// Mitsubishi GX Works2 project: main_01   PLC: FX3U/FX3UC

PROGRAM MAIN
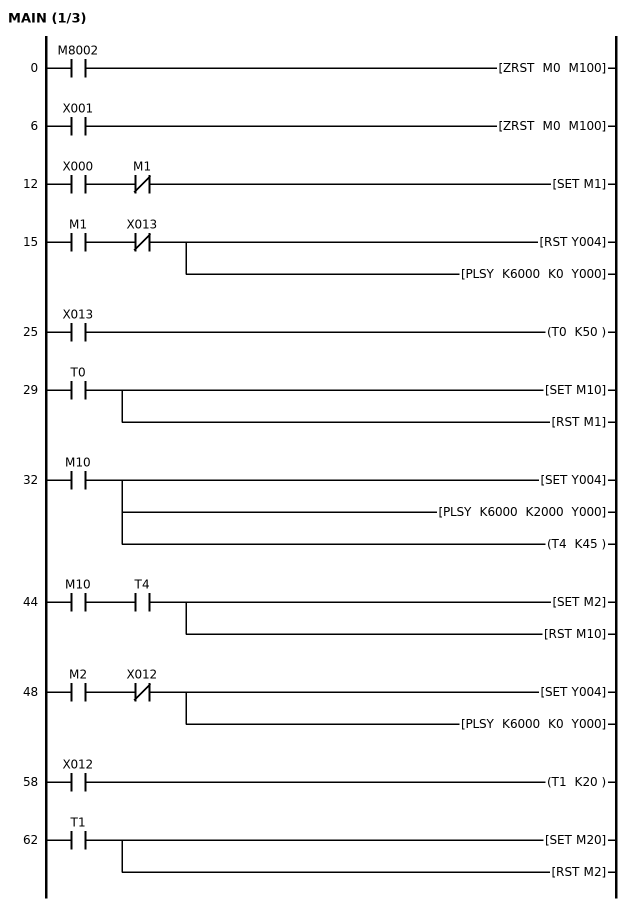
0     LD      M8002
      ZRST    M0 M100
6     LD      X001
      ZRST    M0 M100
12    LD      X000
      ANI     M1
      SET     M1
15    LD      M1
      ANI     X013
      RST     Y004
      PLSY    K6000 K0 Y000
25    LD      X013
      OUT     T0 K50
29    LD      T0
      SET     M10
      RST     M1
32    LD      M10
      SET     Y004
      PLSY    K6000 K2000 Y000
      OUT     T4 K45
44    LD      M10
      AND     T4
      SET     M2
      RST     M10
48    LD      M2
      ANI     X012
      SET     Y004
      PLSY    K6000 K0 Y000
58    LD      X012
      OUT     T1 K20
62    LD      T1
      SET     M20
      RST     M2
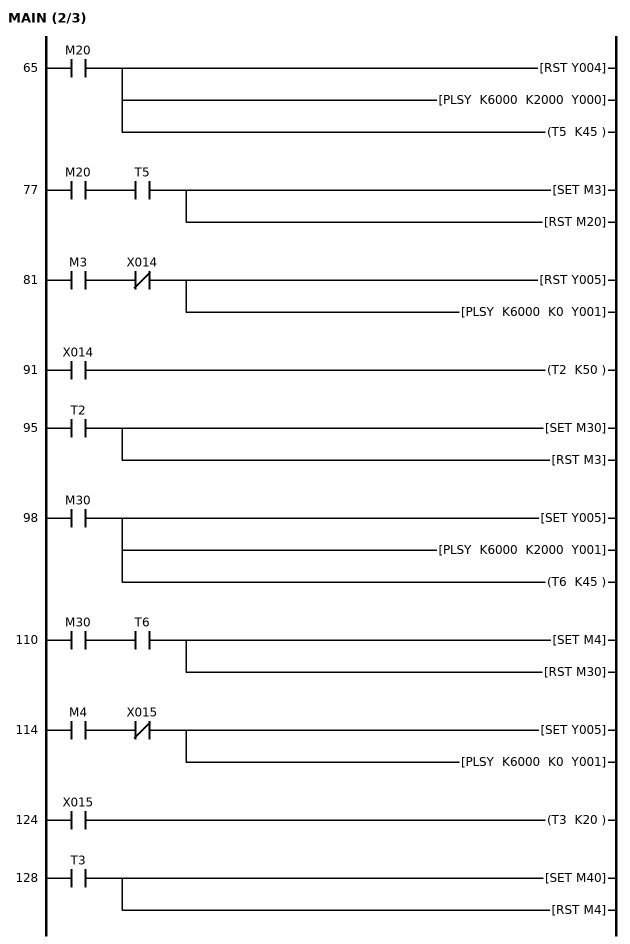
65    LD      M20
      RST     Y004
      PLSY    K6000 K2000 Y000
      OUT     T5 K45
77    LD      M20
      AND     T5
      SET     M3
      RST     M20
81    LD      M3
      ANI     X014
      RST     Y005
      PLSY    K6000 K0 Y001
91    LD      X014
      OUT     T2 K50
95    LD      T2
      SET     M30
      RST     M3
98    LD      M30
      SET     Y005
      PLSY    K6000 K2000 Y001
      OUT     T6 K45
110   LD      M30
      AND     T6
      SET     M4
      RST     M30
114   LD      M4
      ANI     X015
      SET     Y005
      PLSY    K6000 K0 Y001
124   LD      X015
      OUT     T3 K20
128   LD      T3
      SET     M40
      RST     M4
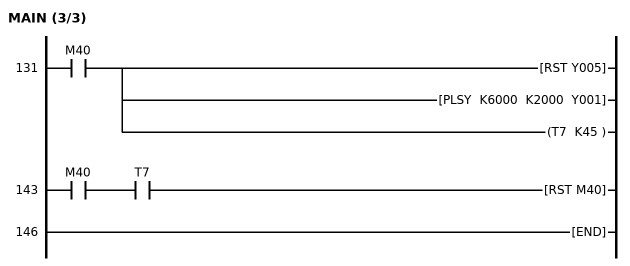
131   LD      M40
      RST     Y005
      PLSY    K6000 K2000 Y001
      OUT     T7 K45
143   LD      M40
      AND     T7
      RST     M40
146   END
END_PROGRAM
